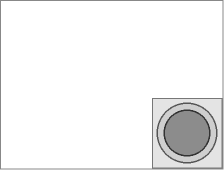
VISUALIZATION resetbtn  // 224x170
    PushSwitch (152,98 70x70), variable: .I_Reset_HMI, behaviour: TAP, style: Switch-PushSwitch-Gray
END_VISUALIZATION

(* stored: Version 1.1.0.1, ProductVersion 3.1.4018.2
   Visu resetbtn: Id {48b2fbdc-024a-4123-bf3b-48145c5852aa} *)
